// TIA Portal project "md_tarikul_islam_sheam(Batch_04)_roll_25_sorting" (V18)

(* hardware
DEVICE "S7-1500/ET200MP station_1"  S7-1500 station
   slot 0: "Rail_0"  Rack  6ES7 590-1***0-0AA0
   slot 1: "PLC_1"  CPU 1516-3 PN/DP  6ES7 516-3AN02-0AB0  V2.9
      slot 3: "CPU display_1"  6ES7591-1BA00-0AA0
      slot 32768: "PROFINET interface_1"  X1
      slot 33024: "PROFINET interface_2"  X2
      slot 33280: "DP interface_1"  X3
      slot 34817: "Virtual CP interface port_1"  Virtual CP interface port  Virtual CP interface port
   slot 2: "DI 32x24VDC HF_1"  DI 32x24VDC HF  6ES7 521-1BL00-0AB0  V2.2
   slot 3: "DQ 32x24VDC/0.5A HF_1"  DQ 32x24VDC/0.5A HF  6ES7 522-1BL01-0AB0  V1.1
   slot 4: "AI 8xU/I/RTD/TC ST_1"  AI 8xU/I/RTD/TC ST  6ES7 531-7KF00-0AB0  V2.2
   slot 5: "AQ 4xU/I ST_1"  AQ 4xU/I ST  6ES7 532-5HD00-0AB0  V2.2
DEVICE "HMI_1"  TP700 Comfort
   slot 0: "HMI_1"  TP700 Comfort  6AV2 124-0GC01-0AX0  17.0.0.0
   slot 1: "HMI_RT_1"  TP700 Comfort  6AV2 124-0GC01-0AX0  17.0.0.0
   slot 5: "HMI_1.IE_CP_1"  PROFINET Interface  17.0.0.0
      slot 1: "PROFINET Interface_1"  PROFINET Interface
         slot 1: "Port_1"  Port
         slot 2: "Port_2"  Port
   slot 7: "HMI_1.MPI/DP_CP_1"  MPI/DP Interface  17.0.0.0
*)

// ===== PLC "PLC_1"  CPU 1516-3 PN/DP =====

VAR_GLOBAL   // PLC tag table "Default tag table"
   "wp_begainning" AT %I0.0 : Bool;
   "conveyor_motor_fwd" AT %Q0.0 : Bool;
   "chute_full" AT %I0.2 : Bool;
   "start" AT %M7.0 : Bool;
   "stop" AT %M9.5 : Bool;
   "chutefull_led" AT %Q1.1 : Bool;
   "def1_ext" AT %I0.1 : Bool;
   "def2_ext" AT %I0.3 : Bool;
   "wp_detect" AT %I0.4 : Bool;
   "optical" AT %I0.5 : Bool;
   "Diffuse" AT %I0.6 : Bool;
   "exteded_def1" AT %Q0.1 : Bool;
   "ext_def2" AT %Q0.2 : Bool;
   "ret_stopper" AT %Q0.3 : Bool;
   "conv_on" AT %M6.0 : Bool;
   "ret_stopper_memory" AT %M6.1 : Bool;
   "def1_adv" AT %M6.2 : Bool;
   "def2_adv" AT %M6.3 : Bool;
   "r_end" AT %M6.4 : Bool;
   "black" AT %M6.5 : Bool;
   "red" AT %M6.6 : Bool;
   "silver" AT %M6.7 : Bool;
   "wp_detected" AT %M1.1 : Bool;
   "reset_rly" AT %M3.1 : Bool;
   "em_relay" AT %M4.0 : Bool;
   "Tag_1" AT %M4.4 : Bool;
   "Tag_2" AT %M5.0 : Bool;
   "Start_led" AT %Q1.0 : Bool;
   "Q2_led" AT %Q1.3 : Bool;
   "reset _Led" AT %Q1.2 : Bool;
   "Tag_5" AT %I2.0 : Bool;
   "RESET" AT %I1.3 : Bool;
   "Start_sw" AT %I1.0 : Bool;
   "Stop_sw" AT %I1.1 : Bool;
END_VAR

ORGANIZATION_BLOCK "Main"   // OB1, LAD, ProgramCycle
TITLE = "Main Program Sweep (Cycle)"
{ S7_Optimized_Access := 'TRUE' }
VERSION : 0.1
   VAR_INPUT
      Initial_Call : Bool;   // Initial call of this OB
      Remanence : Bool;   // =True, if remanent data are available
   END_VAR
BEGIN

REGION Network 1
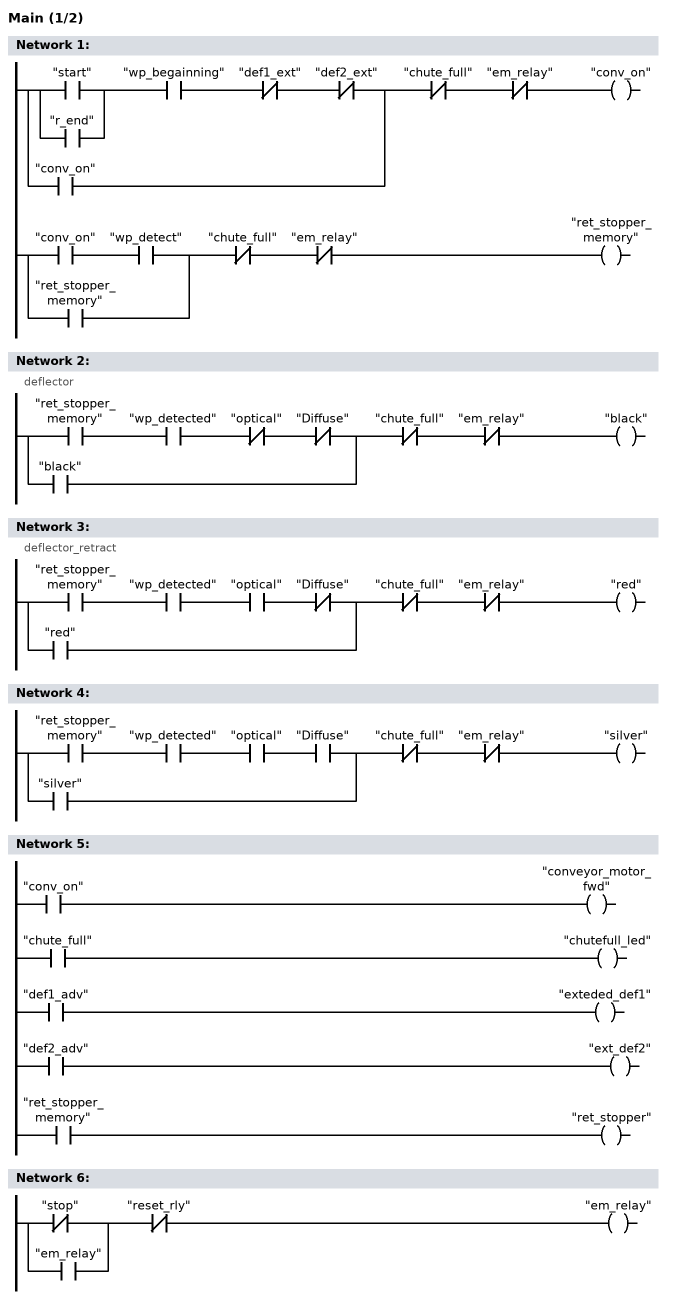
   RUNG wire#powerrail
      Contact( "start" )
      wire#w1
      Contact( "wp_begainning" )
      I_Contact( "def1_ext" )
      I_Contact( "def2_ext" )
      wire#w2
      I_Contact( "chute_full" )
      I_Contact( "em_relay" )
      Coil( "conv_on" )
   END_RUNG
   RUNG wire#powerrail
      Contact( "r_end" )
   END_RUNG wire#w1
   RUNG wire#powerrail
      Contact( "conv_on" )
   END_RUNG wire#w2
   RUNG wire#powerrail
      Contact( "conv_on" )
      Contact( "wp_detect" )
      wire#w3
      I_Contact( "chute_full" )
      I_Contact( "em_relay" )
      Coil( "ret_stopper_memory" )
   END_RUNG
   RUNG wire#powerrail
      Contact( "ret_stopper_memory" )
   END_RUNG wire#w3
   // the same network as SCL:
   "conv_on" := ((("start" OR "r_end") AND "wp_begainning" AND NOT "def1_ext" AND NOT "def2_ext") OR "conv_on") AND NOT "chute_full" AND NOT "em_relay";
   "ret_stopper_memory" := (("conv_on" AND "wp_detect") OR "ret_stopper_memory") AND NOT "chute_full" AND NOT "em_relay";
END_REGION

REGION Network 2
   // deflector
   RUNG wire#powerrail
      Contact( "ret_stopper_memory" )
      Contact( "wp_detected" )
      I_Contact( "optical" )
      I_Contact( "Diffuse" )
      wire#w1
      I_Contact( "chute_full" )
      I_Contact( "em_relay" )
      Coil( "black" )
   END_RUNG
   RUNG wire#powerrail
      Contact( "black" )
   END_RUNG wire#w1
   // the same network as SCL:
   "black" := (("ret_stopper_memory" AND "wp_detected" AND NOT "optical" AND NOT "Diffuse") OR "black") AND NOT "chute_full" AND NOT "em_relay";
END_REGION

REGION Network 3
   // deflector_retract
   RUNG wire#powerrail
      Contact( "ret_stopper_memory" )
      Contact( "wp_detected" )
      Contact( "optical" )
      I_Contact( "Diffuse" )
      wire#w1
      I_Contact( "chute_full" )
      I_Contact( "em_relay" )
      Coil( "red" )
   END_RUNG
   RUNG wire#powerrail
      Contact( "red" )
   END_RUNG wire#w1
   // the same network as SCL:
   "red" := (("ret_stopper_memory" AND "wp_detected" AND "optical" AND NOT "Diffuse") OR "red") AND NOT "chute_full" AND NOT "em_relay";
END_REGION

REGION Network 4
   RUNG wire#powerrail
      Contact( "ret_stopper_memory" )
      Contact( "wp_detected" )
      Contact( "optical" )
      Contact( "Diffuse" )
      wire#w1
      I_Contact( "chute_full" )
      I_Contact( "em_relay" )
      Coil( "silver" )
   END_RUNG
   RUNG wire#powerrail
      Contact( "silver" )
   END_RUNG wire#w1
   // the same network as SCL:
   "silver" := (("ret_stopper_memory" AND "wp_detected" AND "optical" AND "Diffuse") OR "silver") AND NOT "chute_full" AND NOT "em_relay";
END_REGION

REGION Network 5
   RUNG wire#powerrail
      Contact( "conv_on" )
      Coil( "conveyor_motor_fwd" )
   END_RUNG
   RUNG wire#powerrail
      Contact( "chute_full" )
      Coil( "chutefull_led" )
   END_RUNG
   RUNG wire#powerrail
      Contact( "def1_adv" )
      Coil( "exteded_def1" )
   END_RUNG
   RUNG wire#powerrail
      Contact( "def2_adv" )
      Coil( "ext_def2" )
   END_RUNG
   RUNG wire#powerrail
      Contact( "ret_stopper_memory" )
      Coil( "ret_stopper" )
   END_RUNG
   // the same network as SCL:
   "conveyor_motor_fwd" := "conv_on";
   "chutefull_led" := "chute_full";
   "exteded_def1" := "def1_adv";
   "ext_def2" := "def2_adv";
   "ret_stopper" := "ret_stopper_memory";
END_REGION

REGION Network 6
   RUNG wire#powerrail
      I_Contact( "stop" )
      wire#w1
      I_Contact( "reset_rly" )
      Coil( "em_relay" )
   END_RUNG
   RUNG wire#powerrail
      Contact( "em_relay" )
   END_RUNG wire#w1
   // the same network as SCL:
   "em_relay" := (NOT "stop" OR "em_relay") AND NOT "reset_rly";
END_REGION

REGION Network 7
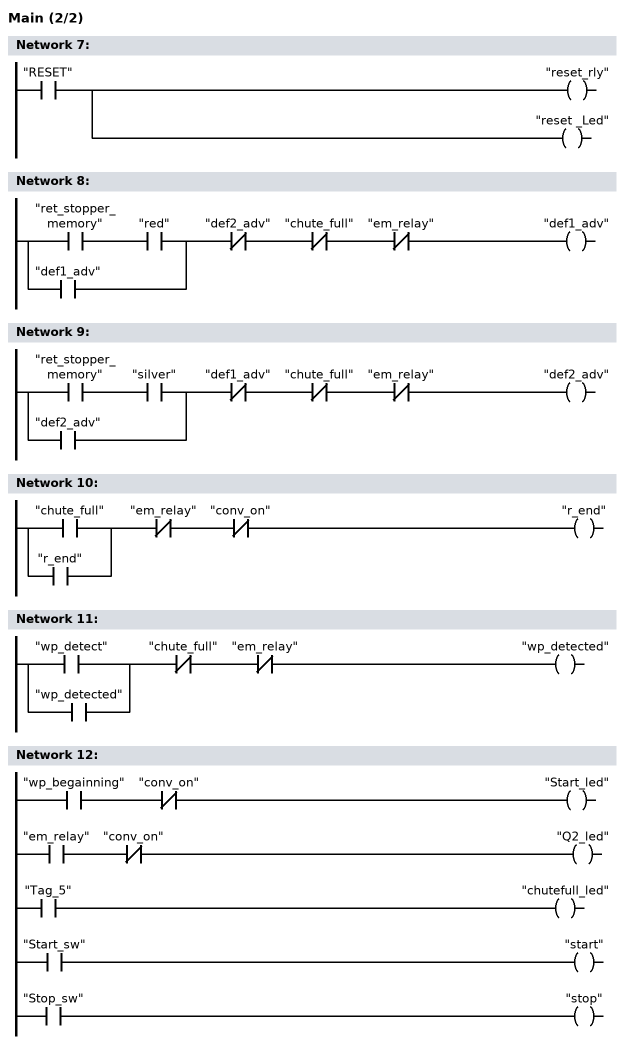
   RUNG wire#powerrail
      Contact( "RESET" )
      wire#w1
      Coil( "reset_rly" )
   END_RUNG
   RUNG wire#w1
      Coil( "reset _Led" )
   END_RUNG
   // the same network as SCL:
   "reset_rly" := "RESET";
   "reset _Led" := "RESET";
END_REGION

REGION Network 8
   RUNG wire#powerrail
      Contact( "ret_stopper_memory" )
      Contact( "red" )
      wire#w1
      I_Contact( "def2_adv" )
      I_Contact( "chute_full" )
      I_Contact( "em_relay" )
      Coil( "def1_adv" )
   END_RUNG
   RUNG wire#powerrail
      Contact( "def1_adv" )
   END_RUNG wire#w1
   // the same network as SCL:
   "def1_adv" := (("ret_stopper_memory" AND "red") OR "def1_adv") AND NOT "def2_adv" AND NOT "chute_full" AND NOT "em_relay";
END_REGION

REGION Network 9
   RUNG wire#powerrail
      Contact( "ret_stopper_memory" )
      Contact( "silver" )
      wire#w1
      I_Contact( "def1_adv" )
      I_Contact( "chute_full" )
      I_Contact( "em_relay" )
      Coil( "def2_adv" )
   END_RUNG
   RUNG wire#powerrail
      Contact( "def2_adv" )
   END_RUNG wire#w1
   // the same network as SCL:
   "def2_adv" := (("ret_stopper_memory" AND "silver") OR "def2_adv") AND NOT "def1_adv" AND NOT "chute_full" AND NOT "em_relay";
END_REGION

REGION Network 10
   RUNG wire#powerrail
      Contact( "chute_full" )
      wire#w1
      I_Contact( "em_relay" )
      I_Contact( "conv_on" )
      Coil( "r_end" )
   END_RUNG
   RUNG wire#powerrail
      Contact( "r_end" )
   END_RUNG wire#w1
   // the same network as SCL:
   "r_end" := ("chute_full" OR "r_end") AND NOT "em_relay" AND NOT "conv_on";
END_REGION

REGION Network 11
   RUNG wire#powerrail
      Contact( "wp_detect" )
      wire#w1
      I_Contact( "chute_full" )
      I_Contact( "em_relay" )
      Coil( "wp_detected" )
   END_RUNG
   RUNG wire#powerrail
      Contact( "wp_detected" )
   END_RUNG wire#w1
   // the same network as SCL:
   "wp_detected" := ("wp_detect" OR "wp_detected") AND NOT "chute_full" AND NOT "em_relay";
END_REGION

REGION Network 12
   RUNG wire#powerrail
      Contact( "wp_begainning" )
      I_Contact( "conv_on" )
      Coil( "Start_led" )
   END_RUNG
   RUNG wire#powerrail
      Contact( "em_relay" )
      I_Contact( "conv_on" )
      Coil( "Q2_led" )
   END_RUNG
   RUNG wire#powerrail
      Contact( "Tag_5" )
      Coil( "chutefull_led" )
   END_RUNG
   RUNG wire#powerrail
      Contact( "Start_sw" )
      Coil( "start" )
   END_RUNG
   RUNG wire#powerrail
      Contact( "Stop_sw" )
      Coil( "stop" )
   END_RUNG
   // the same network as SCL:
   "Start_led" := "wp_begainning" AND NOT "conv_on";
   "Q2_led" := "em_relay" AND NOT "conv_on";
   "chutefull_led" := "Tag_5";
   "start" := "Start_sw";
   "stop" := "Stop_sw";
END_REGION
END_ORGANIZATION_BLOCK

(* ===== HMI "HMI_RT_1" =====
system functions are stored by id; their names below are inferred from use
connection "HMI_Connection_1": ETHERNET, S7_1500_OMS

HMI tags "Default tag table"
   "start" : Bool = PLC start AT %M7.0, 1 s
   "reset" : Bool = PLC RESET AT %I1.3, 1 s
   "r_def1_adv" : Bool = PLC def1_adv AT %M6.2, 1 s
   "r_def2_adv" : Bool = PLC def2_adv AT %M6.3, 1 s
   "r_red" : Bool = PLC red AT %M6.6, 1 s
   "r_silver" : Bool = PLC silver AT %M6.7, 1 s
   "r_black" : Bool = PLC black AT %M6.5, 1 s
   "BLACK_SHOWING" : Bool = PLC BLACK_SHOWING AT %M9.0, 1 s
   "stop" : Bool = PLC stop AT %M9.5, 1 s

Template "Template_1" 800x480
   Button "Exit" at 720,420 size 78x58; TextOff 'Exit'; PictureOff "ExitRuntime_TP700_Comfort_TR"; PictureOn "ExitRuntime_TP700_Comfort_TR"
      on Release: StopRuntime(0)
   Button "Template_Button" at 640,420 size 78x58; TextOff 'Text'
   Button "Template_Button_1" at 560,420 size 78x58; TextOff 'Text'
   Button "Template_Button_2" at 480,420 size 78x58; TextOff 'Text'
   Button "Template_Button_3" at 400,420 size 78x58; TextOff 'Text'
   Button "Template_Button_4" at 321,420 size 78x58; TextOff 'Text'
   Button "Template_Button_5" at 241,420 size 78x58; TextOff 'Text'
   Button "Template_Button_6" at 161,420 size 78x58; TextOff 'Text'
   Button "Template_Button_7" at 81,420 size 78x58; TextOff 'Text'
   Button "Start screen" at 1,420 size 78x58; TextOff 'Start screen'; PictureOff "NavigateHome_TP700_Comfort_TR"; PictureOn "NavigateHome_TP700_Comfort_TR"
      on Release: ActivateScreen("sorting station", 0)

screen "sorting station" 800x480, template "Template_1"
   Button "Button_1" at 369,152 size 96x47; TextOff 'START'
      on Press: function_b14e0dd5("start", 0)
   Button "Button_2" at 371,212 size 96x47; TextOff 'Stop'
      on Press: function_b14e0dd5("stop", 0)
   TextField "Text field_1" at 369,73 size 125x23; Text 'Sorting_Task'
*)